// TIA Portal project "BarcodeScannerPLC" (V12)

(* hardware
DEVICE "S7-1200 station_1"  SIMATIC 1200-Station
   slot 0: "S7-1200 rack"  Rack  V1.0
   slot 1: "PLC_1"  CPU 1212C DC/DC/Rly  6ES7 212-1HD30-0XB0  V2.2
*)

// ===== PLC "PLC_1"  CPU 1212C DC/DC/Rly =====

VAR_GLOBAL   // PLC tag table "Default tag table"
   "DI02" AT %I0.1 : Bool;
   "DI01" AT %I0.0 : Bool;
   "AI01" AT %IW64 : Int;
   "Tag_1" AT %I0.2 : Bool;
   "Tag_2" AT %I0.3 : Bool;
   "DO01" AT %Q0.0 : Bool;
   "DO02" AT %Q0.1 : Bool;
   "Counter1" AT %MW0 : Int;
   "Counter2" AT %MW2 : Int;
   "AI01Scaled" AT %MD10 : Real;
   "CounterAI" AT %M12.0 : Bool;
   "Watchdog" AT %M100.0 : Bool;
   "WatchdogOutput" AT %M100.1 : Bool;
END_VAR

DATA_BLOCK "DB1"   // DB1
{ S7_Optimized_Access := 'FALSE' }
VERSION : 0.1
   VAR
      Machine1Motor : Bool;
      Machine2Motor : Bool;
      Machine1Counter : Int := 0;
      Machine2Counter : Int;
      Machine1ResetCounter : Bool;
      Machine2ResetCounter : Bool;
      CorrectBarcodeScanCounter2 : Int;
      StartButton1 : Bool;
      StopButton1 : Bool;
      BlankLight1 : Bool;
      MissedLight1 : Bool;
      Machine1Counter1 : Int;
      Machine1Counter2 : Int;
      Machine2Counter1 : Int;
      Machine2Counter2 : Int;
   END_VAR
BEGIN
END_DATA_BLOCK

// folder: System blocks/Program resources

DATA_BLOCK "Machine01Counter1"   // DB2
{ S7_Optimized_Access := 'FALSE' }
AUTHOR : Simatic
FAMILY : IEC
NAME : CNTR
VERSION : 1.0
// stored: InstanceOfName ?
"?"
BEGIN
END_DATA_BLOCK

DATA_BLOCK "Machine02Counter2"   // DB3
{ S7_Optimized_Access := 'FALSE' }
AUTHOR : Simatic
FAMILY : IEC
NAME : CNTR
VERSION : 1.0
// stored: InstanceOfName ?
"?"
BEGIN
END_DATA_BLOCK

DATA_BLOCK "IEC_Timer_0_DB"   // DB4
{ S7_Optimized_Access := 'FALSE' }
AUTHOR : Simatic
FAMILY : IEC
NAME : IEC_TMR
VERSION : 1.0
// stored: InstanceOfName ?
"?"
BEGIN
END_DATA_BLOCK

// folder: (top level)

FUNCTION "StopMachine2When" : Void   // FC1, SCL
{ S7_Optimized_Access := 'FALSE' }
VERSION : 0.1
BEGIN
   IF ("DB1".Machine2Counter - "DB1".CorrectBarcodeScanCounter2)>2 THEN
     "DB1".Machine2Motor:=true;
     "DB1".CorrectBarcodeScanCounter2:="DB1".Machine2Counter;
   END_IF;
END_FUNCTION

ORGANIZATION_BLOCK "Main"   // OB1, LAD, ProgramCycle
TITLE = "Main Program Sweep (Cycle)"
{ S7_Optimized_Access := 'FALSE' }
VERSION : 0.1
BEGIN
END_ORGANIZATION_BLOCK